PROGRAM PRG_PMPS
VAR
END_VAR

END_PROGRAM

(* stored: Version 1.1.0.1, ProductVersion 3.1.4022.16
   POU PRG_PMPS: Id {3bbd9cd5-72c9-4b35-aa2f-63d3e3610a6e}, SpecialFunc None *)
